SUBAPPLICATION Gesamtzaehler (* Subapplication Type *)
  (* Standard: 61499-2 *)
  (* Version 1.0, 2023-02-17, Franz *)
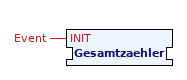
  EVENT_INPUT
    INIT; (* Initialization Request *)
  END_EVENT
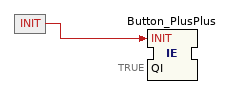
  FBS
    Button_PlusPlus : IE(QI := TRUE);
  END_FBS
  EVENT_CONNECTIONS
    INIT TO Button_PlusPlus.INIT;
  END_CONNECTIONS
END_SUBAPPLICATION
